// TIA Portal project "ProgettoIniziale" (V17)

(* hardware
DEVICE "Stazione S7-1500/ET200MP_1"  S7-1500 station
   slot 0: "Telaio di montaggio_0"  Rack  6ES7 590-1***0-0AA0
   slot 1: "PLC_1"  CPU 1511-1 PN  6ES7 511-1AK02-0AB0  V2.9
      slot 3: "Display CPU_1"  6ES7591-1AA00-0AA0
      slot 32768: "Interfaccia PROFINET_1"  X1
         slot 32769: "Porta_1"  X1 P1
         slot 32770: "Porta_2"  X1 P2
      slot 34817: "Virtual CP interface port_1"  Virtual CP interface port  Virtual CP interface port
*)

// ===== PLC "PLC_1"  CPU 1511-1 PN =====

ORGANIZATION_BLOCK "Main"   // OB1, LAD, ProgramCycle
TITLE = "Main Program Sweep (Cycle)"
{ S7_Optimized_Access := 'TRUE' }
VERSION : 0.1
   VAR_INPUT
      Initial_Call : Bool;   // Initial call of this OB
      Remanence : Bool;   // =True, if remanent data are available
   END_VAR
BEGIN
END_ORGANIZATION_BLOCK

// ===== library: MasterCopy "Motore" =====

FUNCTION_BLOCK "Motore"   // FB1, LAD
{ S7_Optimized_Access := 'TRUE' }
VERSION : 0.1
   VAR_INPUT
      Enable : Bool;
      Setpoint : Real;
   END_VAR
   VAR_OUTPUT
      VelAttuale : Real;
   END_VAR
BEGIN
END_FUNCTION_BLOCK